(* CODESYS project SW_DMU218_3091.library
   Author: Leuze electronic GmbH + Co. KG
   Placeholder: DMU218_3091
   Title: DMU218_3091
   Version: 1.0.0
   Description: IO-Link service function blocks library
   Company: Leuze electronic GmbH + Co. KG

Project tree, tasks and I/O mapping:
  libraries: Tc2_Standard, * (Beckhoff Automation GmbH); Tc2_System, * (Beckhoff Automation GmbH); Tc2_Utilities, * (Beckhoff Automation GmbH)
  Leuze/
    DMU218_3091/
      data type ST_Leuze_IOL_AnalogRange_Data
      data type ST_Leuze_IOL_AnalogRange_Selection
      data type ST_Leuze_IOL_Commands_Data
      data type ST_Leuze_IOL_Commands_Selection
      data type ST_Leuze_IOL_Data
      data type ST_Leuze_IOL_DeviceAccessLocks_Data
      data type ST_Leuze_IOL_DeviceAccessLocks_Selection
      data type ST_Leuze_IOL_DirectParametersPage1_Data
      data type ST_Leuze_IOL_DirectParametersPage1_Selection
      data type ST_Leuze_IOL_DirectParametersPage2_Data
      data type ST_Leuze_IOL_DirectParametersPage2_Selection
      data type ST_Leuze_IOL_Network_Data
      data type ST_Leuze_IOL_Network_Selection
      data type ST_Leuze_IOL_ProcessDataLimits_Data
      data type ST_Leuze_IOL_ProcessDataLimits_Selection
      data type ST_Leuze_IOL_Selection
      data type ST_Leuze_IOL_Setpoints_Data
      data type ST_Leuze_IOL_Setpoints_Selection
      data type ST_Leuze_IOL_SwitchpointBdc1_Data
      data type ST_Leuze_IOL_SwitchpointBdc1_Selection
      data type ST_Leuze_IOL_TeachpointSp1_Data
      data type ST_Leuze_IOL_TeachpointSp1_Selection
      data type ST_Leuze_IOL_TeachpointSp2_Data
      data type ST_Leuze_IOL_TeachpointSp2_Selection
      data type ST_Leuze_IOL_TeachState_Data
      data type ST_Leuze_IOL_TeachState_Selection
    Internal/
      function F_Leuze_IOL_GetArrayT [ST]
      function F_Leuze_IOL_GetBoolean [ST]
      function F_Leuze_IOL_GetByteLength [ST]
      function F_Leuze_IOL_GetInteger [ST]
      function F_Leuze_IOL_GetRecordT [ST]
      function F_Leuze_IOL_GetString [ST]
      function F_Leuze_IOL_SetArrayT [ST]
      function F_Leuze_IOL_SetBoolean [ST]
      function F_Leuze_IOL_SetInteger [ST]
      function F_Leuze_IOL_SetRecordT [ST]
      function F_Leuze_IOL_SetString [ST]
      function F_Leuze_IOL_SortComplex [ST]
      function block FB_Leuze_IOL_AdsReadWrite [ST]
      data type ST_Leuze_IOL_CommandQueue
      data type ST_Leuze_IOL_Error
    function F_Leuze_PD_DMU218_3091 [ST]
    function block FB_Leuze_IOL_DMU218_3091 [ST]
    data type ST_Leuze_IOL_DMU218_3091
    data type ST_Leuze_PD_DMU218_3091
*)

// Leuze/DMU218_3091/ST_Leuze_IOL_AnalogRange_Data
TYPE ST_Leuze_IOL_AnalogRange_Data :
STRUCT     // [READ_WRITE]
	nLowerLimit : UINT := 150;    // [READ_WRITE]
	nUpperLimit : UINT := 1500;    // [READ_WRITE]
END_STRUCT
END_TYPE

// Leuze/DMU218_3091/ST_Leuze_IOL_AnalogRange_Selection
TYPE ST_Leuze_IOL_AnalogRange_Selection :
STRUCT     // [READ_WRITE]
	bAll : BOOL;    // [READ_WRITE] all parameters of complex data type
	bLowerLimit : BOOL;    // [READ_WRITE]
	bUpperLimit : BOOL;    // [READ_WRITE]
END_STRUCT
END_TYPE

// Leuze/DMU218_3091/ST_Leuze_IOL_Commands_Data
TYPE ST_Leuze_IOL_Commands_Data :
STRUCT     // [WRITE_ONLY] Command interface for applications. A positive acknowledge indicates the complete and correct finalization of the requested function.
	nCmdRestoreFactorySettings : UINT := 130;    // [WRITE_ONLY] Restore Factory Settings
	nCmdTeachApply : UINT := 64;    // [WRITE_ONLY] Teach Apply
	nCmdSetpoint1SingleValueTeach : UINT := 65;    // [WRITE_ONLY] Setpoint 1 Single Value Teach
	nCmdSetpoint2SingleValueTeach : UINT := 66;    // [WRITE_ONLY] Setpoint 2 Single Value Teach
	nCmdTwoValueTeachTp1Sp1 : UINT := 67;    // [WRITE_ONLY] Two Value Teach TP1 SP1
	nCmdTwoValueTeachTp2Sp1 : UINT := 68;    // [WRITE_ONLY] Two Value Teach TP2 SP1
	nCmdTwoValueTeachTp1Sp2 : UINT := 69;    // [WRITE_ONLY] Two Value Teach TP1 SP2
	nCmdTwoValueTeachTp2Sp2 : UINT := 70;    // [WRITE_ONLY] Two Value Teach TP2 SP2
	nCmdSetpoint1DynamicTeachStart : UINT := 71;    // [WRITE_ONLY] Setpoint 1 Dynamic Teach Start
	nCmdSetpoint1DynamicTeachStop : UINT := 72;    // [WRITE_ONLY] Setpoint 1 Dynamic Teach Stop
	nCmdSetpoint2DynamicTeachStart : UINT := 73;    // [WRITE_ONLY] Setpoint 2 Dynamic Teach Start
	nCmdSetpoint2DynamicTeachStop : UINT := 74;    // [WRITE_ONLY] Setpoint 2 Dynamic Teach Stop
	nCmdTeachCancel : UINT := 79;    // [WRITE_ONLY] Teach Cancel
	nCmdSetAnalogOutputLowerLimit : UINT := 161;    // [WRITE_ONLY] Set Analog Output Lower Limit
	nCmdSetAnalogOutputUpperLimit : UINT := 162;    // [WRITE_ONLY] Set Analog Output Upper Limit
	nCmdResetDiagnosisInformation : UINT := 163;    // [WRITE_ONLY] Reset Diagnosis Information
	nCmdStopMeasurement : UINT := 164;    // [WRITE_ONLY] Stop measurement
	nCmdStartMeasurement : UINT := 165;    // [WRITE_ONLY] Start measurement
	nCmdSingleMeasurement : UINT := 166;    // [WRITE_ONLY] Single measurement
	nCmdIoLink11SystemTestCommand240Event8DfeAppears : UINT := 240;    // [WRITE_ONLY] IO-Link 1.1 system test command 240, Event 8DFE appears
	nCmdIoLink11SystemTestCommand241Event8DfeDisappears : UINT := 241;    // [WRITE_ONLY] IO-Link 1.1 system test command 241, Event 8DFE disappears
	nCmdIoLink11SystemTestCommand242Event8DffAppears : UINT := 242;    // [WRITE_ONLY] IO-Link 1.1 system test command 242, Event 8DFF appears
	nCmdIoLink11SystemTestCommand243Event8DffDisappears : UINT := 243;    // [WRITE_ONLY] IO-Link 1.1 system test command 243, Event 8DFF disappears
END_STRUCT
END_TYPE

// Leuze/DMU218_3091/ST_Leuze_IOL_Commands_Selection
TYPE ST_Leuze_IOL_Commands_Selection :
STRUCT     // [WRITE_ONLY] Command interface for applications. A positive acknowledge indicates the complete and correct finalization of the requested function.
	bCmdRestoreFactorySettings : BOOL;    // [WRITE_ONLY] Restore Factory Settings
	bCmdTeachApply : BOOL;    // [WRITE_ONLY] Teach Apply
	bCmdSetpoint1SingleValueTeach : BOOL;    // [WRITE_ONLY] Setpoint 1 Single Value Teach
	bCmdSetpoint2SingleValueTeach : BOOL;    // [WRITE_ONLY] Setpoint 2 Single Value Teach
	bCmdTwoValueTeachTp1Sp1 : BOOL;    // [WRITE_ONLY] Two Value Teach TP1 SP1
	bCmdTwoValueTeachTp2Sp1 : BOOL;    // [WRITE_ONLY] Two Value Teach TP2 SP1
	bCmdTwoValueTeachTp1Sp2 : BOOL;    // [WRITE_ONLY] Two Value Teach TP1 SP2
	bCmdTwoValueTeachTp2Sp2 : BOOL;    // [WRITE_ONLY] Two Value Teach TP2 SP2
	bCmdSetpoint1DynamicTeachStart : BOOL;    // [WRITE_ONLY] Setpoint 1 Dynamic Teach Start
	bCmdSetpoint1DynamicTeachStop : BOOL;    // [WRITE_ONLY] Setpoint 1 Dynamic Teach Stop
	bCmdSetpoint2DynamicTeachStart : BOOL;    // [WRITE_ONLY] Setpoint 2 Dynamic Teach Start
	bCmdSetpoint2DynamicTeachStop : BOOL;    // [WRITE_ONLY] Setpoint 2 Dynamic Teach Stop
	bCmdTeachCancel : BOOL;    // [WRITE_ONLY] Teach Cancel
	bCmdSetAnalogOutputLowerLimit : BOOL;    // [WRITE_ONLY] Set Analog Output Lower Limit
	bCmdSetAnalogOutputUpperLimit : BOOL;    // [WRITE_ONLY] Set Analog Output Upper Limit
	bCmdResetDiagnosisInformation : BOOL;    // [WRITE_ONLY] Reset Diagnosis Information
	bCmdStopMeasurement : BOOL;    // [WRITE_ONLY] Stop measurement
	bCmdStartMeasurement : BOOL;    // [WRITE_ONLY] Start measurement
	bCmdSingleMeasurement : BOOL;    // [WRITE_ONLY] Single measurement
	bCmdIoLink11SystemTestCommand240Event8DfeAppears : BOOL;    // [WRITE_ONLY] IO-Link 1.1 system test command 240, Event 8DFE appears
	bCmdIoLink11SystemTestCommand241Event8DfeDisappears : BOOL;    // [WRITE_ONLY] IO-Link 1.1 system test command 241, Event 8DFE disappears
	bCmdIoLink11SystemTestCommand242Event8DffAppears : BOOL;    // [WRITE_ONLY] IO-Link 1.1 system test command 242, Event 8DFF appears
	bCmdIoLink11SystemTestCommand243Event8DffDisappears : BOOL;    // [WRITE_ONLY] IO-Link 1.1 system test command 243, Event 8DFF disappears
END_STRUCT
END_TYPE

// Leuze/DMU218_3091/ST_Leuze_IOL_Data
TYPE ST_Leuze_IOL_Data :
STRUCT 
	stCommands : ST_Leuze_IOL_Commands_Data;
	stDirectParametersPage1 : ST_Leuze_IOL_DirectParametersPage1_Data;
	stDirectParametersPage2 : ST_Leuze_IOL_DirectParametersPage2_Data;
	nSystemCommand : UINT;    // [WRITE_ONLY] Command interface for applications. A positive acknowledge indicates the complete and correct finalization of the requested function.
	stDeviceAccessLocks : ST_Leuze_IOL_DeviceAccessLocks_Data;
	sVendorName : STRING := 'Leuze electronic GmbH + Co. KG';    // [READ_ONLY] The vendor name that is assigned to a Vendor ID.
	sVendorText : STRING := 'The Sensor People';    // [READ_ONLY] Additional information about the vendor.
	sProductName : STRING;    // [READ_ONLY] Complete product name.
	sProductId : STRING;    // [READ_ONLY] Vendor-specific product or type identification (e.g., item number or model number).
	sProductText : STRING;    // [READ_ONLY] Additional product information for the device.
	sFirmwareRevision : STRING;    // [READ_ONLY] Unique, vendor-specific identifier of the firmware revision of the individual device.
	sApplicationSpecificTag : STRING;    // [READ_WRITE] Possibility to mark a device with user- or application-specific information.
	nErrorCount : UINT;    // [READ_ONLY] Number of errors that occurred in the technology-specific application since power on or restart.
	nDeviceStatus : UINT;    // [READ_ONLY] Indicator for the current device condition and diagnosis state.
	stTeachState : ST_Leuze_IOL_TeachState_Data;
	stSetpoints : ST_Leuze_IOL_Setpoints_Data;
	stSwitchpointBdc1 : ST_Leuze_IOL_SwitchpointBdc1_Data;
	sLot : STRING;    // [READ_ONLY] production lot
	nOnDelaySwitchingOutput : UINT := 0;    // [READ_WRITE] on delay for the binary data channel
	nOffDelaySwitchingOutput : UINT := 0;    // [READ_WRITE] off delay for the binary data channel
	nMultiIOPin4 : UINT := 0;    // [READ_WRITE] polarity of the switching output
	nMultiIOPin2 : UINT := 2;    // [READ_WRITE] operation mode for Multi I/O (Pin 2)
	stAnalogRange : ST_Leuze_IOL_AnalogRange_Data;
	nTemperatureCompensation : UINT := 0;    // [READ_WRITE]
	stTeachpointSp1 : ST_Leuze_IOL_TeachpointSp1_Data;
	stTeachpointSp2 : ST_Leuze_IOL_TeachpointSp2_Data;
	stProcessDataLimits : ST_Leuze_IOL_ProcessDataLimits_Data;
	nSwitchCounter : UINT := 0;    // [READ_ONLY] number of switching after power-up or reset
	nTemperatureInternal : INT;    // [READ_ONLY] Sensor temperature
	stNetwork : ST_Leuze_IOL_Network_Data;
END_STRUCT
END_TYPE

// Leuze/DMU218_3091/ST_Leuze_IOL_DeviceAccessLocks_Data
TYPE ST_Leuze_IOL_DeviceAccessLocks_Data :
STRUCT     // [READ_WRITE] The access to the device parameters can be restricted by setting appropriate flags within this parameter.
	bParameterWriteAccess : BOOL := 0;    // [READ_WRITE] This lock prevents the write access to all read/write parameters of the device except for the parameter 'Device Access Locks'.
	bDataStorage : BOOL;    // [READ_WRITE] This lock prevents the write access to the device parameters via the data storage mechanism.
	bLocalParameterization : BOOL := 0;    // [READ_WRITE] This lock prevents the device settings from being changed via local operating elements on the device.
	bLocalUserInterface : BOOL;    // [READ_WRITE] This lock prevents the access to the device settings and display via a local user interface. The user interface is disabled.
END_STRUCT
END_TYPE

// Leuze/DMU218_3091/ST_Leuze_IOL_DeviceAccessLocks_Selection
TYPE ST_Leuze_IOL_DeviceAccessLocks_Selection :
STRUCT     // [READ_WRITE] The access to the device parameters can be restricted by setting appropriate flags within this parameter.
	bAll : BOOL;    // [READ_WRITE] all parameters of complex data type
END_STRUCT
END_TYPE

// Leuze/DMU218_3091/ST_Leuze_IOL_DirectParametersPage1_Data
TYPE ST_Leuze_IOL_DirectParametersPage1_Data :
STRUCT     // [READ_WRITE] Comprises the required parameters defining the communication characteristics and identifiers for device validation.
	nReserved_1 : UINT;    // [READ_ONLY] ; Suffix "_1" (parameter index or subindex) added because of duplicate parameter names.
	nMasterCycleTime : UINT;    // [READ_ONLY] Communication: Current communication cycle duration used by the master. This value defines the process data cycle.
	nMinCycleTime : UINT;    // [READ_ONLY] Communication: Minimum communication cycle duration supported by the device. This value defines the lowest possible process data cycle.
	nMSequenceCapability : UINT;    // [READ_ONLY] Communication: Information on the structure and the supported features of the communication messages.
	nIoLinkRevisionId : UINT := 17;    // [READ_ONLY] Communication: Identifier for the currently used communication protocol revision.
	nProcessDataInputLength : UINT;    // [READ_ONLY] Communication: Information on width and features of the process input data (Process Data from Device to Master).
	nProcessDataOutputLength : UINT;    // [READ_ONLY] Communication: Information on width of the process output data (Process Data from Master to Device).
	nVendorId1 : UINT;    // [READ_ONLY] Identification: Highest octet of the Vendor ID. Combined with the parameter Vendor ID 2, this parameter defines the 16-bit value of the unique Vendor ID as assigned by the IO-Link Community.
	nVendorId2 : UINT;    // [READ_ONLY] Identification: Lowest octet of the Vendor ID. Combined with the parameter Vendor ID 1, this parameter defines the 16-bit value of the unique Vendor ID as assigned by the IO-Link Community.
	nDeviceId1 : UINT;    // [READ_ONLY] Identification: Highest octet of the Device ID. Combined with the parameters Device ID 2 and 3, this parameter defines the 24-bit value of the vendor-specific Device ID.
	nDeviceId2 : UINT;    // [READ_ONLY] Identification: Middle octet of the Device ID. Combined with the parameters Device ID 1 and 3, this parameter defines the 24-bit value of the vendor-specific Device ID.
	nDeviceId3 : UINT;    // [READ_ONLY] Identification: Lowest octet of the Device ID. Combined with the parameters Device ID 1 and 2, this parameter defines the 24-bit value of the vendor-specific Device ID.
	nReserved_13 : UINT;    // [READ_ONLY] ; Suffix "_13" (parameter index or subindex) added because of duplicate parameter names.
	nReserved_14 : UINT;    // [READ_ONLY] ; Suffix "_14" (parameter index or subindex) added because of duplicate parameter names.
	nReserved_15 : UINT;    // [READ_ONLY] ; Suffix "_15" (parameter index or subindex) added because of duplicate parameter names.
	nSystemCommand : UINT;    // [WRITE_ONLY] Application: Command interface for devices without ISDU support. Validity and execution of commands are not confirmed.
END_STRUCT
END_TYPE

// Leuze/DMU218_3091/ST_Leuze_IOL_DirectParametersPage1_Selection
TYPE ST_Leuze_IOL_DirectParametersPage1_Selection :
STRUCT     // [READ_WRITE] Comprises the required parameters defining the communication characteristics and identifiers for device validation.
	bAll : BOOL;    // [READ_WRITE] all parameters of complex data type
	bReserved_1 : BOOL;    // [READ_ONLY] ; Suffix "_1" (parameter index or subindex) added because of duplicate parameter names.
	bMasterCycleTime : BOOL;    // [READ_ONLY] Communication: Current communication cycle duration used by the master. This value defines the process data cycle.
	bMinCycleTime : BOOL;    // [READ_ONLY] Communication: Minimum communication cycle duration supported by the device. This value defines the lowest possible process data cycle.
	bMSequenceCapability : BOOL;    // [READ_ONLY] Communication: Information on the structure and the supported features of the communication messages.
	bIoLinkRevisionId : BOOL;    // [READ_ONLY] Communication: Identifier for the currently used communication protocol revision.
	bProcessDataInputLength : BOOL;    // [READ_ONLY] Communication: Information on width and features of the process input data (Process Data from Device to Master).
	bProcessDataOutputLength : BOOL;    // [READ_ONLY] Communication: Information on width of the process output data (Process Data from Master to Device).
	bVendorId1 : BOOL;    // [READ_ONLY] Identification: Highest octet of the Vendor ID. Combined with the parameter Vendor ID 2, this parameter defines the 16-bit value of the unique Vendor ID as assigned by the IO-Link Community.
	bVendorId2 : BOOL;    // [READ_ONLY] Identification: Lowest octet of the Vendor ID. Combined with the parameter Vendor ID 1, this parameter defines the 16-bit value of the unique Vendor ID as assigned by the IO-Link Community.
	bDeviceId1 : BOOL;    // [READ_ONLY] Identification: Highest octet of the Device ID. Combined with the parameters Device ID 2 and 3, this parameter defines the 24-bit value of the vendor-specific Device ID.
	bDeviceId2 : BOOL;    // [READ_ONLY] Identification: Middle octet of the Device ID. Combined with the parameters Device ID 1 and 3, this parameter defines the 24-bit value of the vendor-specific Device ID.
	bDeviceId3 : BOOL;    // [READ_ONLY] Identification: Lowest octet of the Device ID. Combined with the parameters Device ID 1 and 2, this parameter defines the 24-bit value of the vendor-specific Device ID.
	bReserved_13 : BOOL;    // [READ_ONLY] ; Suffix "_13" (parameter index or subindex) added because of duplicate parameter names.
	bReserved_14 : BOOL;    // [READ_ONLY] ; Suffix "_14" (parameter index or subindex) added because of duplicate parameter names.
	bReserved_15 : BOOL;    // [READ_ONLY] ; Suffix "_15" (parameter index or subindex) added because of duplicate parameter names.
	bSystemCommand : BOOL;    // [WRITE_ONLY] Application: Command interface for devices without ISDU support. Validity and execution of commands are not confirmed.
END_STRUCT
END_TYPE

// Leuze/DMU218_3091/ST_Leuze_IOL_DirectParametersPage2_Data
TYPE ST_Leuze_IOL_DirectParametersPage2_Data :
STRUCT     // [READ_WRITE] A set of parameters for devices without ISDU support.
	nDeviceSpecificParameter1 : UINT;    // [READ_WRITE]
	nDeviceSpecificParameter2 : UINT;    // [READ_WRITE]
	nDeviceSpecificParameter3 : UINT;    // [READ_WRITE]
	nDeviceSpecificParameter4 : UINT;    // [READ_WRITE]
	nDeviceSpecificParameter5 : UINT;    // [READ_WRITE]
	nDeviceSpecificParameter6 : UINT;    // [READ_WRITE]
	nDeviceSpecificParameter7 : UINT;    // [READ_WRITE]
	nDeviceSpecificParameter8 : UINT;    // [READ_WRITE]
	nDeviceSpecificParameter9 : UINT;    // [READ_WRITE]
	nDeviceSpecificParameter10 : UINT;    // [READ_WRITE]
	nDeviceSpecificParameter11 : UINT;    // [READ_WRITE]
	nDeviceSpecificParameter12 : UINT;    // [READ_WRITE]
	nDeviceSpecificParameter13 : UINT;    // [READ_WRITE]
	nDeviceSpecificParameter14 : UINT;    // [READ_WRITE]
	nDeviceSpecificParameter15 : UINT;    // [READ_WRITE]
	nDeviceSpecificParameter16 : UINT;    // [READ_WRITE]
END_STRUCT
END_TYPE

// Leuze/DMU218_3091/ST_Leuze_IOL_DirectParametersPage2_Selection
TYPE ST_Leuze_IOL_DirectParametersPage2_Selection :
STRUCT     // [READ_WRITE] A set of parameters for devices without ISDU support.
	bAll : BOOL;    // [READ_WRITE] all parameters of complex data type
	bDeviceSpecificParameter1 : BOOL;    // [READ_WRITE]
	bDeviceSpecificParameter2 : BOOL;    // [READ_WRITE]
	bDeviceSpecificParameter3 : BOOL;    // [READ_WRITE]
	bDeviceSpecificParameter4 : BOOL;    // [READ_WRITE]
	bDeviceSpecificParameter5 : BOOL;    // [READ_WRITE]
	bDeviceSpecificParameter6 : BOOL;    // [READ_WRITE]
	bDeviceSpecificParameter7 : BOOL;    // [READ_WRITE]
	bDeviceSpecificParameter8 : BOOL;    // [READ_WRITE]
	bDeviceSpecificParameter9 : BOOL;    // [READ_WRITE]
	bDeviceSpecificParameter10 : BOOL;    // [READ_WRITE]
	bDeviceSpecificParameter11 : BOOL;    // [READ_WRITE]
	bDeviceSpecificParameter12 : BOOL;    // [READ_WRITE]
	bDeviceSpecificParameter13 : BOOL;    // [READ_WRITE]
	bDeviceSpecificParameter14 : BOOL;    // [READ_WRITE]
	bDeviceSpecificParameter15 : BOOL;    // [READ_WRITE]
	bDeviceSpecificParameter16 : BOOL;    // [READ_WRITE]
END_STRUCT
END_TYPE

// Leuze/DMU218_3091/ST_Leuze_IOL_Network_Data
TYPE ST_Leuze_IOL_Network_Data :
STRUCT     // [READ_WRITE]
	nRoleInNetwork : UINT := 0;    // [READ_WRITE]
	nDeviceNoMasterHighestNo : UINT := 1;    // [READ_WRITE]
END_STRUCT
END_TYPE

// Leuze/DMU218_3091/ST_Leuze_IOL_Network_Selection
TYPE ST_Leuze_IOL_Network_Selection :
STRUCT     // [READ_WRITE]
	bAll : BOOL;    // [READ_WRITE] all parameters of complex data type
	bRoleInNetwork : BOOL;    // [READ_WRITE]
	bDeviceNoMasterHighestNo : BOOL;    // [READ_WRITE]
END_STRUCT
END_TYPE

// Leuze/DMU218_3091/ST_Leuze_IOL_ProcessDataLimits_Data
TYPE ST_Leuze_IOL_ProcessDataLimits_Data :
STRUCT     // [READ_ONLY] Process data limit values
	nLower : UINT;    // [READ_ONLY] lower limit after power-up or reset
	nUpper : UINT;    // [READ_ONLY] upper limit after power-up or reset
END_STRUCT
END_TYPE

// Leuze/DMU218_3091/ST_Leuze_IOL_ProcessDataLimits_Selection
TYPE ST_Leuze_IOL_ProcessDataLimits_Selection :
STRUCT     // [READ_ONLY] Process data limit values
	bAll : BOOL;    // [READ_ONLY] all parameters of complex data type
	bLower : BOOL;    // [READ_ONLY] lower limit after power-up or reset
	bUpper : BOOL;    // [READ_ONLY] upper limit after power-up or reset
END_STRUCT
END_TYPE

// Leuze/DMU218_3091/ST_Leuze_IOL_Selection
TYPE ST_Leuze_IOL_Selection :
STRUCT 
	stCommands : ST_Leuze_IOL_Commands_Selection;
	stDirectParametersPage1 : ST_Leuze_IOL_DirectParametersPage1_Selection;
	stDirectParametersPage2 : ST_Leuze_IOL_DirectParametersPage2_Selection;
	bSystemCommand : BOOL;    // [WRITE_ONLY] Command interface for applications. A positive acknowledge indicates the complete and correct finalization of the requested function.
	stDeviceAccessLocks : ST_Leuze_IOL_DeviceAccessLocks_Selection;
	bVendorName : BOOL;    // [READ_ONLY] The vendor name that is assigned to a Vendor ID.
	bVendorText : BOOL;    // [READ_ONLY] Additional information about the vendor.
	bProductName : BOOL;    // [READ_ONLY] Complete product name.
	bProductId : BOOL;    // [READ_ONLY] Vendor-specific product or type identification (e.g., item number or model number).
	bProductText : BOOL;    // [READ_ONLY] Additional product information for the device.
	bFirmwareRevision : BOOL;    // [READ_ONLY] Unique, vendor-specific identifier of the firmware revision of the individual device.
	bApplicationSpecificTag : BOOL;    // [READ_WRITE] Possibility to mark a device with user- or application-specific information.
	bErrorCount : BOOL;    // [READ_ONLY] Number of errors that occurred in the technology-specific application since power on or restart.
	bDeviceStatus : BOOL;    // [READ_ONLY] Indicator for the current device condition and diagnosis state.
	stTeachState : ST_Leuze_IOL_TeachState_Selection;
	stSetpoints : ST_Leuze_IOL_Setpoints_Selection;
	stSwitchpointBdc1 : ST_Leuze_IOL_SwitchpointBdc1_Selection;
	bLot : BOOL;    // [READ_ONLY] production lot
	bOnDelaySwitchingOutput : BOOL;    // [READ_WRITE] on delay for the binary data channel
	bOffDelaySwitchingOutput : BOOL;    // [READ_WRITE] off delay for the binary data channel
	bMultiIOPin4 : BOOL;    // [READ_WRITE] polarity of the switching output
	bMultiIOPin2 : BOOL;    // [READ_WRITE] operation mode for Multi I/O (Pin 2)
	stAnalogRange : ST_Leuze_IOL_AnalogRange_Selection;
	bTemperatureCompensation : BOOL;    // [READ_WRITE]
	stTeachpointSp1 : ST_Leuze_IOL_TeachpointSp1_Selection;
	stTeachpointSp2 : ST_Leuze_IOL_TeachpointSp2_Selection;
	stProcessDataLimits : ST_Leuze_IOL_ProcessDataLimits_Selection;
	bSwitchCounter : BOOL;    // [READ_ONLY] number of switching after power-up or reset
	bTemperatureInternal : BOOL;    // [READ_ONLY] Sensor temperature
	stNetwork : ST_Leuze_IOL_Network_Selection;
END_STRUCT
END_TYPE

// Leuze/DMU218_3091/ST_Leuze_IOL_Setpoints_Data
TYPE ST_Leuze_IOL_Setpoints_Data :
STRUCT     // [READ_WRITE] threshold measurement value of a sensor for the edge of a binary output signal 1
	nParam1Bdc1Q1 : UINT := 150;    // [READ_WRITE] threshold measurement value
	nParam2Bdc1Q1 : UINT := 1500;    // [READ_WRITE] threshold measurement value
END_STRUCT
END_TYPE

// Leuze/DMU218_3091/ST_Leuze_IOL_Setpoints_Selection
TYPE ST_Leuze_IOL_Setpoints_Selection :
STRUCT     // [READ_WRITE] threshold measurement value of a sensor for the edge of a binary output signal 1
	bAll : BOOL;    // [READ_WRITE] all parameters of complex data type
	bParam1Bdc1Q1 : BOOL;    // [READ_WRITE] threshold measurement value
	bParam2Bdc1Q1 : BOOL;    // [READ_WRITE] threshold measurement value
END_STRUCT
END_TYPE

// Leuze/DMU218_3091/ST_Leuze_IOL_SwitchpointBdc1_Data
TYPE ST_Leuze_IOL_SwitchpointBdc1_Data :
STRUCT     // [READ_WRITE] mode, logic and hysteresis for binary data channel 1
	nLogic : UINT := 0;    // [READ_WRITE] switching information is transmitted in inverted or not inverted manner
	nMode : UINT := 2;    // [READ_WRITE] operation mode for binary signal
	nHysteresis : UINT := 2;    // [READ_WRITE]
END_STRUCT
END_TYPE

// Leuze/DMU218_3091/ST_Leuze_IOL_SwitchpointBdc1_Selection
TYPE ST_Leuze_IOL_SwitchpointBdc1_Selection :
STRUCT     // [READ_WRITE] mode, logic and hysteresis for binary data channel 1
	bAll : BOOL;    // [READ_WRITE] all parameters of complex data type
	bLogic : BOOL;    // [READ_WRITE] switching information is transmitted in inverted or not inverted manner
	bMode : BOOL;    // [READ_WRITE] operation mode for binary signal
	bHysteresis : BOOL;    // [READ_WRITE]
END_STRUCT
END_TYPE

// Leuze/DMU218_3091/ST_Leuze_IOL_TeachpointSp1_Data
TYPE ST_Leuze_IOL_TeachpointSp1_Data :
STRUCT     // [READ_ONLY] Values detected during teach
	nTp1 : UINT;    // [READ_ONLY] detected lower limit during teach-in procedure
	nTp2 : UINT;    // [READ_ONLY] detected upper limit during teach-in procedure
END_STRUCT
END_TYPE

// Leuze/DMU218_3091/ST_Leuze_IOL_TeachpointSp1_Selection
TYPE ST_Leuze_IOL_TeachpointSp1_Selection :
STRUCT     // [READ_ONLY] Values detected during teach
	bAll : BOOL;    // [READ_ONLY] all parameters of complex data type
	bTp1 : BOOL;    // [READ_ONLY] detected lower limit during teach-in procedure
	bTp2 : BOOL;    // [READ_ONLY] detected upper limit during teach-in procedure
END_STRUCT
END_TYPE

// Leuze/DMU218_3091/ST_Leuze_IOL_TeachpointSp2_Data
TYPE ST_Leuze_IOL_TeachpointSp2_Data :
STRUCT     // [READ_ONLY] Values detected during teach
	nTp1 : UINT;    // [READ_ONLY] detected lower limit during teach-in procedure
	nTp2 : UINT;    // [READ_ONLY] detected upper limit during teach-in procedure
END_STRUCT
END_TYPE

// Leuze/DMU218_3091/ST_Leuze_IOL_TeachpointSp2_Selection
TYPE ST_Leuze_IOL_TeachpointSp2_Selection :
STRUCT     // [READ_ONLY] Values detected during teach
	bAll : BOOL;    // [READ_ONLY] all parameters of complex data type
	bTp1 : BOOL;    // [READ_ONLY] detected lower limit during teach-in procedure
	bTp2 : BOOL;    // [READ_ONLY] detected upper limit during teach-in procedure
END_STRUCT
END_TYPE

// Leuze/DMU218_3091/ST_Leuze_IOL_TeachState_Data
TYPE ST_Leuze_IOL_TeachState_Data :
STRUCT     // [READ_ONLY] indication of the current state of the teach-in procedure and teach point setting
	nTeachState : UINT := 0;    // [READ_ONLY] indication of the current state of the teach-in procedure
END_STRUCT
END_TYPE

// Leuze/DMU218_3091/ST_Leuze_IOL_TeachState_Selection
TYPE ST_Leuze_IOL_TeachState_Selection :
STRUCT     // [READ_ONLY] indication of the current state of the teach-in procedure and teach point setting
	bAll : BOOL;    // [READ_ONLY] all parameters of complex data type
END_STRUCT
END_TYPE

// Leuze/Internal/ST_Leuze_IOL_CommandQueue
TYPE ST_Leuze_IOL_CommandQueue :
STRUCT
	nIndex : INT;		// Index of parameter in queue
    nSubIndex : INT;	// SubIndex of a parameter in queue
    nBitLength : UINT;	// Bit length of a parameter
END_STRUCT
END_TYPE

// Leuze/Internal/ST_Leuze_IOL_Error
TYPE ST_Leuze_IOL_Error :
STRUCT
    nBlockError : WORD;			// Error number representing FB where error occured 
	nAdsReadError : UDINT;		// ADS read error code
	nAdsWriteError : UDINT;		// ADS write error code
	nIndex : INT;				// IO-Link index to which the error code refers
	nSubIndex : INT;			// IO-Link sub-index to which the error code refers
END_STRUCT
END_TYPE

// Leuze/ST_Leuze_IOL_DMU218_3091
TYPE ST_Leuze_IOL_DMU218_3091 :
STRUCT
	stSelection : ST_Leuze_IOL_Selection;
	stData : ST_Leuze_IOL_Data;
END_STRUCT
END_TYPE

// Leuze/ST_Leuze_PD_DMU218_3091
TYPE ST_Leuze_PD_DMU218_3091 :
STRUCT
	nMeasuredValue : UINT;
	bSwitchStateBdc1Q1 : BOOL;
END_STRUCT
END_TYPE

// Leuze/Internal/F_Leuze_IOL_GetArrayT
FUNCTION F_Leuze_IOL_GetArrayT : BOOL
VAR_INPUT
	nArraySize : UINT;
    nItemPosition : UINT;
    nBitLength : UINT;
END_VAR
VAR_IN_OUT 
      aIolRecords : ARRAY[0..cNUMBER_IOLINK_DATA] OF BYTE;
      aTempItems : ARRAY[0..cNUMBER_IOLINK_DATA] OF BYTE;
END_VAR
VAR
      nTempArrayByteLength : UINT;
      nTempStartByte : UINT;
      nTempStartBit : UINT;
      nTempIolBitLength : UINT;
      nTempIolByteLength : UINT;
      nTempIndex : UINT;
      nTempShiftByte : BYTE;
      bTempByteFill : BOOL;
END_VAR
VAR CONSTANT 
	  cNUMBER_IOLINK_DATA : UINT := 255;   //   Number of IO Link record data
	  cBITS_IN_BYTE : UINT := 8;   //   Number of bits in byte
END_VAR

// =============================================================================
// Name:    IO-Link internal function 
//          Array data type - Integer, Bool
// Date:    01.01.2021
// ==============================================================================

// Initialize variables
	bTempByteFill := FALSE;
	
// Bit length of the current item
	nTempIolBitLength := nBitLength;
	
// Get byte length of the current item
	nTempIolByteLength := F_Leuze_IOL_GetByteLength(nTempIolBitLength);
	
// Get byte length of the whole array
	nTempArrayByteLength := F_Leuze_IOL_GetByteLength(nArraySize);
	
	
// Calculate the start byte of the current array item
	nTempStartByte := nTempArrayByteLength - 1 - ((nArraySize - (nItemPosition * nTempIolBitLength)) / cBITS_IN_BYTE);
	
// Calculate the start bit of the current array item
	nTempStartBit := (nArraySize - (nItemPosition * nTempIolBitLength)) MOD cBITS_IN_BYTE;
	
// Calculate index
	nTempIndex := nTempIolByteLength - 1;
	
// Get array item
	WHILE nTempIolBitLength > 0 DO
		IF NOT bTempByteFill THEN	    
			IF (nTempIolBitLength + nTempStartBit) < cBITS_IN_BYTE THEN
				nTempShiftByte := SHL(aIolRecords[nTempStartByte], cBITS_IN_BYTE - (nTempIolBitLength + nTempStartBit));
				nTempShiftByte := SHR(nTempShiftByte, cBITS_IN_BYTE - nTempIolBitLength);
			ELSE
				nTempShiftByte := SHR(aIolRecords[nTempStartByte], nTempStartBit);
			END_IF;
			
			aTempItems[nTempIndex] := nTempShiftByte;
			
			IF (nTempStartBit + nTempIolBitLength) = cBITS_IN_BYTE THEN
				nTempStartByte := nTempStartByte - 1;
			END_IF;
			
			IF (nTempStartBit + nTempIolBitLength) > cBITS_IN_BYTE THEN
				nTempStartByte := nTempStartByte - 1;
				bTempByteFill := TRUE;
			ELSE
				nTempIndex := nTempIndex - 1;
			END_IF;
			
			nTempIolBitLength := nTempIolBitLength - (cBITS_IN_BYTE - nTempStartBit);
		ELSE	   
	    IF nTempStartBit >= nTempIolBitLength THEN
			nTempShiftByte := SHL(aIolRecords[nTempStartByte], cBITS_IN_BYTE - nTempIolBitLength);
			nTempShiftByte := SHR(nTempShiftByte, nTempStartBit - nTempIolBitLength);
	    ELSE
	    	nTempShiftByte := SHL(aIolRecords[nTempStartByte], cBITS_IN_BYTE - nTempStartBit);
	    END_IF;
	    
	    aTempItems[nTempIndex] := nTempShiftByte XOR aTempItems[nTempIndex];	    
	    nTempIolBitLength := nTempIolBitLength - nTempStartBit;
	    nTempIndex := nTempIndex - 1;
	    bTempByteFill := FALSE;
		END_IF;
	END_WHILE;

END_FUNCTION

// Leuze/Internal/F_Leuze_IOL_GetByteLength
FUNCTION F_Leuze_IOL_GetByteLength : UINT
VAR_INPUT
	nBitLength: UINT;
END_VAR
VAR
	nByteLength: UINT;
END_VAR

VAR CONSTANT
	cBITS_IN_BYTE: UINT := 8;
END_VAR

nByteLength := nBitLength / cBITS_IN_BYTE;
IF NOT (nBitLength MOD cBITS_IN_BYTE = 0) THEN
		nByteLength := nByteLength + 1;
END_IF;
F_Leuze_IOL_GetByteLength := nByteLength;

END_FUNCTION

// Leuze/Internal/F_Leuze_IOL_GetBoolean
FUNCTION F_Leuze_IOL_GetBoolean : BOOL
VAR_INPUT 
      nComplex : INT;	// Data type: cBASIC_TYPE, cCOMPLEX_RECORD_TYPE, cCOMPLEX_ARRAY_TYPE
      nComplexDataTypeSize : INT;	// Record or Array type size
      nOffset : INT;	// Bit Offset
   END_VAR
   VAR_IN_OUT 
      aIolRecords : ARRAY[0..cNUMBER_IOLINK_DATA] OF BYTE;
      aTempItems : ARRAY[0..cNUMBER_IOLINK_DATA] OF BYTE;
   END_VAR
   VAR CONSTANT 
      cNUMBER_IOLINK_DATA : INT := 255;   //   Number of IO Link record data
      cBASIC_TYPE : INT := 0;
      cCOMPLEX_RECORD_TYPE : INT := 1;
      cCOMPLEX_ARRAY_TYPE : INT := 2;
   END_VAR

// =============================================================================
// Name:    IO-Link internal function 
//  		GetBoolean
// Date:    01.07.2020
// ==============================================================================
	
// Data type is part of a Record data type
IF nComplex = cCOMPLEX_RECORD_TYPE THEN		
  F_Leuze_IOL_GetRecordT(nComplexDataTypeSize, nOffset, 1, aIolRecords, aTempItems);
  // Data type is part of a Array data type
ELSIF nComplex = cCOMPLEX_ARRAY_TYPE THEN
  F_Leuze_IOL_GetArrayT(INT_TO_UINT(nComplexDataTypeSize), INT_TO_UINT(nOffset), 1, aIolRecords, aTempItems);
END_IF;
	
// In a nComplex data type the coding of booleans are only 1 bit wide. There is no padding to byte 
IF nComplex > cBASIC_TYPE THEN
  IF aTempItems[0].0 = 1 THEN
    F_Leuze_IOL_GetBoolean := TRUE;
  ELSE
    F_Leuze_IOL_GetBoolean := FALSE;
  END_IF;
ELSE
  IF aIolRecords[0] > 16#00 THEN
    F_Leuze_IOL_GetBoolean := TRUE;
  ELSE
    F_Leuze_IOL_GetBoolean := FALSE;
  END_IF;
END_IF;

END_FUNCTION

// Leuze/Internal/F_Leuze_IOL_GetRecordT
FUNCTION F_Leuze_IOL_GetRecordT : BOOL
VAR_INPUT 
      nRecordSize : INT;
      nBitOffset : INT;
      nBitLength : INT;
   END_VAR
   VAR_IN_OUT 
      aIolRecords : ARRAY[0..cNUMBER_IOLINK_DATA] OF BYTE;
      aTempItems : ARRAY[0..cNUMBER_IOLINK_DATA] OF BYTE;
   END_VAR
   VAR
      nTempStartByte : INT;
      nTempStartBit : Int;
      tempIOLBitLength : Int;
      tempIOLByteLength : Int;
      nTempIndex : Int;
      nTempShiftByte : Byte;
      bTempByteFill : Bool;
   END_VAR
   VAR CONSTANT 
	  cNUMBER_IOLINK_DATA : INT := 255;   //   Number of IO Link record data
	  cBITS_IN_BYTE : INT := 8;   //   Number of bits in byte
   END_VAR

// =============================================================================
// Name:    IO-Link internal function 
//    		Record data type - Integer, Bool
// Date:    01.07.2020
// ==============================================================================
	
// Initialize variables
	bTempByteFill := FALSE;
	
// Bit length of the current item
	tempIOLBitLength := nBitLength;
	
// Get byte length of the current item
	tempIOLByteLength := tempIOLBitLength / cBITS_IN_BYTE;
	IF NOT (tempIOLBitLength MOD cBITS_IN_BYTE = 0) THEN
		tempIOLByteLength := tempIOLByteLength + 1;
	END_IF;
		
// Calculate the start byte of the current item
	nTempStartByte := (nRecordSize / cBITS_IN_BYTE) - 1 - (nBitOffset / cBITS_IN_BYTE);
	IF NOT(nRecordSize MOD cBITS_IN_BYTE = 0) THEN
		nTempStartByte := nTempStartByte +1;
	END_IF;

// Calculate the start bit of the current item
	nTempStartBit := nBitOffset MOD cBITS_IN_BYTE;
	
// Calculate index
	nTempIndex := tempIOLByteLength - 1;
	
// Get record item
	WHILE tempIOLBitLength > 0 DO
		IF NOT bTempByteFill THEN		
			IF (tempIOLBitLength + nTempStartBit) < cBITS_IN_BYTE THEN
				nTempShiftByte := SHL(aIolRecords[nTempStartByte], INT_TO_UINT(cBITS_IN_BYTE - (tempIOLBitLength + nTempStartBit)));
				nTempShiftByte := SHR(nTempShiftByte, INT_TO_UINT(cBITS_IN_BYTE - tempIOLBitLength));
			ELSE
				nTempShiftByte := SHR(aIolRecords[nTempStartByte], INT_TO_UINT(nTempStartBit));
			END_IF;
			aTempItems[nTempIndex] := nTempShiftByte;
			
			IF (nTempStartBit + tempIOLBitLength) = cBITS_IN_BYTE THEN
				nTempStartByte := nTempStartByte - 1;
			END_IF;
			
			IF (nTempStartBit + tempIOLBitLength) > cBITS_IN_BYTE THEN
				nTempStartByte := nTempStartByte - 1;
				bTempByteFill := TRUE;
			ELSE
				nTempIndex := nTempIndex - 1;
			END_IF;
			
			tempIOLBitLength := tempIOLBitLength - (cBITS_IN_BYTE - nTempStartBit);
		ELSE		
			IF nTempStartBit >= tempIOLBitLength THEN
				nTempShiftByte := SHL(aIolRecords[nTempStartByte], INT_TO_UINT(cBITS_IN_BYTE - tempIOLBitLength));
				nTempShiftByte := SHR(nTempShiftByte, INT_TO_UINT(nTempStartBit - tempIOLBitLength));
			ELSE
				nTempShiftByte := SHL(aIolRecords[nTempStartByte], INT_TO_UINT(cBITS_IN_BYTE - nTempStartBit));
			END_IF;			
			aTempItems[nTempIndex] := nTempShiftByte XOR aTempItems[nTempIndex];			
			tempIOLBitLength := tempIOLBitLength - nTempStartBit;
			nTempIndex := nTempIndex - 1;
			bTempByteFill := FALSE;
		END_IF;
	END_WHILE;

END_FUNCTION

// Leuze/Internal/F_Leuze_IOL_GetInteger
FUNCTION F_Leuze_IOL_GetInteger : DWORD
VAR_INPUT 
      nComplex : INT;	// Data type: cBASIC_TYPE, cCOMPLEX_RECORD_TYPE, cCOMPLEX_ARRAY_TYPE
      nComplexDataTypeSize : INT;	// Record or Array type size
      nOffset : INT;	// Bit Offset
      nBitLength : INT;
      bIsSigned : BOOL;
   END_VAR
   VAR_IN_OUT 
      aIolRecords : ARRAY[0..cNUMBER_IOLINK_DATA] OF BYTE;
      aTempItems : ARRAY[0..cNUMBER_IOLINK_DATA] OF BYTE;
   END_VAR
VAR
	nTempOutput : DWORD;   
    nTempIndex : INT;
    nTempIolByteLength : INT;
    nTemp : DWORD;
    aTempValues : ARRAY[0..3] OF BYTE;
	pOutput: POINTER TO ARRAY[0..3] OF BYTE;
END_VAR
VAR CONSTANT
	  cNUMBER_IOLINK_DATA : INT := 255;   //   Number of IO Link record data
	  cBITS_IN_BYTE : INT := 8;   //   Number of bits in byte
      cBASIC_TYPE : INT := 0;
      cCOMPLEX_RECORD_TYPE : INT := 1;
      cCOMPLEX_ARRAY_TYPE : INT := 2;
   END_VAR

// =============================================================================
// Name:    IO-Link internal function 
//   		GetInteger
// Date:    01.01.2021
// ==============================================================================

// Data type is part of a Record data type
	IF nComplex = cCOMPLEX_RECORD_TYPE THEN
		F_Leuze_IOL_GetRecordT(nComplexDataTypeSize, nOffset, nBitLength, aIolRecords, aTempItems);
	// Data type is part of a Array data type
	ELSIF nComplex = cCOMPLEX_ARRAY_TYPE THEN
		F_Leuze_IOL_GetArrayT(INT_TO_UINT(nComplexDataTypeSize), INT_TO_UINT(nOffset), INT_TO_UINT(nBitLength), aIolRecords, aTempItems);
	END_IF;
	
// Initialization
	F_Leuze_IOL_GetInteger := 16#00;
	aTempValues[0] := 0;
	aTempValues[1] := 0;
	aTempValues[2] := 0;
	aTempValues[3] := 0;
	
// Get byte length
	nTempIolByteLength := nBitLength / cBITS_IN_BYTE;
	IF NOT (nBitLength MOD cBITS_IN_BYTE = 0) THEN
		nTempIolByteLength := nTempIolByteLength + 1;
	END_IF;
	
// There is no padding to 1,2,4 byte if a nComplex data type is used
	IF (nComplex = cBASIC_TYPE) AND (nTempIolByteLength = 3) THEN
		nTempIolByteLength := 4;
	END_IF;
	
	IF nTempIolByteLength > 0 AND nTempIolByteLength <= 4 THEN
	// Get the value out of the IO-Link Record and change the byte order
	FOR nTempIndex := 0 TO nTempIolByteLength - 1 DO
		IF nComplex > cBASIC_TYPE THEN
			aTempValues[nTempIndex] := aTempItems[nTempIolByteLength - 1 - nTempIndex];
		ELSE
			aTempValues[nTempIndex] := aIolRecords[nTempIolByteLength - 1 - nTempIndex];
		END_IF;
	END_FOR;	  	 
	  	
// Copy result into a DWORD variable
	F_Leuze_IOL_GetInteger := PDWORD_TO_DWORD(ADR(aTempValues));
	  
// Received value can be a negative value
	IF bIsSigned THEN
	// Create a signed value
		IF DWORD_TO_BOOL(SHR(F_Leuze_IOL_GetInteger, INT_TO_UINT(nBitLength) - 1)) THEN
			nTemp := 2;
			FOR nTempIndex := 1 TO nBitLength - 1 DO
				nTemp := nTemp * 2;
			END_FOR;
			F_Leuze_IOL_GetInteger := F_Leuze_IOL_GetInteger OR (16#FFFF_FFFF XOR (nTemp - 1));
			END_IF;
		END_IF;
	END_IF;

END_FUNCTION

// Leuze/Internal/F_Leuze_IOL_GetString
FUNCTION F_Leuze_IOL_GetString : STRING
VAR_INPUT 
      nComplex : INT;	// Data type: cBASIC_TYPE, cCOMPLEX_RECORD_TYPE, cCOMPLEX_ARRAY_TYPE
      nComplexDataTypeSize : INT;	// Record or Array type size
      nOffset : INT;	// Bit Offset
      nFixedLength : INT; // In bits
   END_VAR
   VAR_IN_OUT 
      aIolRecords : ARRAY[0..cNUMBER_IOLINK_DATA] OF BYTE;
      aTempItems : ARRAY[0..cNUMBER_IOLINK_DATA] OF BYTE;
   END_VAR
   VAR 
      nTempIndex : INT;
	  nTempStringLength : UINT;
	  nTempByteLength : INT;
   END_VAR
   VAR CONSTANT 
	cNUMBER_IOLINK_DATA : INT := 255;   //   Number of IO Link record data
	cBITS_IN_BYTE : INT := 8;   //   Number of bits in byte
	cBASIC_TYPE : INT := 0;
	cCOMPLEX_RECORD_TYPE : INT := 1;
	cCOMPLEX_ARRAY_TYPE : INT := 2;
END_VAR

// =============================================================================
	// Name:    IO-Link internal function 
	//          Get string
	// Date:    01.07.2020
	// ==============================================================================	
	//Data type is part of a Record data type
	IF nComplex = cCOMPLEX_RECORD_TYPE THEN
	  F_Leuze_IOL_GetRecordT( nComplexDataTypeSize, nOffset, nFixedLength, aIolRecords, aTempItems);
	//Data type is part of a Array data type
	ELSIF nComplex = cCOMPLEX_ARRAY_TYPE THEN
	  F_Leuze_IOL_GetArrayT(INT_TO_UINT(nComplexDataTypeSize), INT_TO_UINT(nOffset), INT_TO_UINT(nFixedLength), aIolRecords, aTempItems);
	END_IF;
	
	//Initialization
	nTempStringLength := 0;
	nTempByteLength := nFixedLength / cBITS_IN_BYTE;

	//Calculate the actual string length
	IF nTempByteLength <= 232 THEN
	  FOR nTempIndex := 0 TO nTempByteLength - 1 DO
	    IF nComplex > 0 THEN
	      IF aTempItems[nTempIndex] = 16#00 THEN
	        EXIT;
	      ELSE
	        nTempStringLength := nTempStringLength + 1;
	      END_IF;
	    ELSE
	      IF aIolRecords[nTempIndex] = 16#00 THEN
	        EXIT;
	      ELSE
	        nTempStringLength := nTempStringLength + 1;
	      END_IF;
	    END_IF;
	  END_FOR;
	  
	  //Copy to the RETURN value
	  IF nComplex > cBASIC_TYPE THEN		  		   
		  F_Leuze_IOL_GetString := BYTEARR_TO_MAXSTRING(aTempItems);		  
	  ELSE
	    IF nTempStringLength = 0 THEN
	      F_Leuze_IOL_GetString := '';
	    ELSE
			F_Leuze_IOL_GetString := BYTEARR_TO_MAXSTRING(aIolRecords);
	    END_IF;
	  END_IF;
	ELSE
	  F_Leuze_IOL_GetString := '';
	END_IF;

END_FUNCTION

// Leuze/Internal/F_Leuze_IOL_SetArrayT
FUNCTION F_Leuze_IOL_SetArrayT : BOOL
VAR_INPUT 
      nArraySize : UINT;
      nItemPosition : UINT;
      nBitLength : UINT;
   END_VAR
   VAR_IN_OUT 
      aIolRecords : ARRAY[0..cNUMBER_IOLINK_DATA] OF BYTE;
      aTempItems : ARRAY[0..cNUMBER_IOLINK_DATA] OF BYTE;
   END_VAR
   VAR
      nTempArrayByteLength : UINT;
      nTempStartByte : UINT;
      nTempStartBit : UINT;
      nTempIolBitLength : UINT;
      nTempIndex : UINT;
      nTempShiftByte : BYTE;
      bTempByteFill : BOOL;
   END_VAR
   VAR CONSTANT 
	  cNUMBER_IOLINK_DATA : UINT := 255;   //   Number of IO Link record data
	  cBITS_IN_BYTE : UINT := 8;   //   Number of bits in byte
   END_VAR

// =============================================================================
// Name:    IO-Link internal function 
//	 	    Set ArrayT
// Date:    01.01.2021
// ==============================================================================
	
// Initialize variables
	bTempByteFill := FALSE;
	nTempIndex := 0;

// Bit length of the current item
	nTempIolBitLength := nBitLength;

// Get byte length of the whole array
	nTempArrayByteLength := F_Leuze_IOL_GetByteLength(nArraySize);
	
// Calculate the start byte of the current array item
	nTempStartByte := nTempArrayByteLength - 1 - ((nArraySize - (nItemPosition * nTempIolBitLength)) / cBITS_IN_BYTE);
	
// Calculate the start bit of the current array item
	nTempStartBit := (nArraySize - (nItemPosition * nTempIolBitLength)) MOD cBITS_IN_BYTE;
	
// Set array item
	WHILE nTempIolBitLength > 0 DO
	  IF NOT bTempByteFill THEN
	    IF (nTempIolBitLength + nTempStartBit) < cBITS_IN_BYTE THEN
	      nTempShiftByte := SHL(aTempItems[nTempIndex], cBITS_IN_BYTE - nTempIolBitLength);
	      nTempShiftByte := SHR(nTempShiftByte, (cBITS_IN_BYTE - nTempIolBitLength) - nTempStartBit);
	    ELSE
	      nTempShiftByte := SHL(aTempItems[nTempIndex], nTempStartBit);
	    END_IF;
	    
	    aIolRecords[nTempStartByte] := aIolRecords[nTempStartByte] + nTempShiftByte;
	    
	    IF (nTempStartBit + nTempIolBitLength) = cBITS_IN_BYTE THEN
	      nTempStartByte := nTempStartByte - 1;
	    END_IF;
	    
	    IF (nTempStartBit + nTempIolBitLength) > cBITS_IN_BYTE THEN
	      nTempStartByte := nTempStartByte - 1;
	      bTempByteFill := TRUE;
	    ELSE
	      nTempIndex := nTempIndex + 1;
	    END_IF;
	    
	    nTempIolBitLength := nTempIolBitLength - (cBITS_IN_BYTE - nTempStartBit);
	  ELSE
	    IF nTempStartBit > nTempIolBitLength THEN
	      nTempShiftByte := SHL(aTempItems[nTempIndex], nTempStartBit - nTempIolBitLength);
	      nTempShiftByte := SHR(nTempShiftByte, cBITS_IN_BYTE - nTempIolBitLength);
	    ELSE
	      nTempShiftByte := SHR(aTempItems[nTempIndex], cBITS_IN_BYTE - nTempStartBit);
	    END_IF;
	    
	    aIolRecords[nTempStartByte] := aIolRecords[nTempStartByte] + nTempShiftByte;
	    nTempIolBitLength := nTempIolBitLength - nTempStartBit;
	    nTempIndex := nTempIndex + 1;
	    bTempByteFill := FALSE;
	  END_IF;
	END_WHILE;

END_FUNCTION

// Leuze/Internal/F_Leuze_IOL_SetBoolean
FUNCTION F_Leuze_IOL_SetBoolean : BOOL
VAR_INPUT 
      nComplex : INT;	// Data type: cBASIC_TYPE, cCOMPLEX_RECORD_TYPE, cCOMPLEX_ARRAY_TYPE
      nComplexDataTypeSize : INT;	// Record or Array type size
      nOffset : INT;	// Bit Offset
      bSource : BOOL;
   END_VAR
   VAR_IN_OUT 
      aIolRecords : ARRAY[0..cNUMBER_IOLINK_DATA] OF BYTE;
      aTempItems : ARRAY[0..cNUMBER_IOLINK_DATA] OF BYTE;
   END_VAR
   VAR CONSTANT 
      cNUMBER_IOLINK_DATA : INT := 255;   //   Number of IO Link record data
      cBASIC_TYPE : INT := 0;
      cCOMPLEX_RECORD_TYPE : INT := 1;
      cCOMPLEX_ARRAY_TYPE : INT := 2;
   END_VAR

// =============================================================================
// Name:    IO-Link internal function 
//          Set Boolean
// Date:    01.07.2020
// ==============================================================================
// In a nComplex data type the coding of booleans are only 1 bit wide. There is no padding to byte
IF nComplex > cBASIC_TYPE THEN
  IF bSource THEN
    aTempItems[0] := (aTempItems[0] AND 2#1111_1110) + 1;
  ELSE
    aTempItems[0] := aTempItems[0] AND 2#1111_1110;
  END_IF;
ELSE
  IF bSource THEN
    aIolRecords[0] := 16#FF;
  ELSE
    aIolRecords[0] := 16#00;
  END_IF;
END_IF;

// Data type is part of a Record data type
IF nComplex = cCOMPLEX_RECORD_TYPE THEN
  F_Leuze_IOL_SetRecordT(nComplexDataTypeSize, nOffset, 1, aIolRecords, aTempItems);
// Data type is part of a Array data type
ELSIF nComplex = cCOMPLEX_ARRAY_TYPE THEN
  F_Leuze_IOL_SetArrayT(INT_TO_UINT(nComplexDataTypeSize), INT_TO_UINT(nOffset), 1, aIolRecords, aTempItems);
END_IF;

END_FUNCTION

// Leuze/Internal/F_Leuze_IOL_SetRecordT
FUNCTION F_Leuze_IOL_SetRecordT : BOOL
VAR_INPUT 
      nRecordSize : INT;
      nBitOffset : INT;
      nBitLength : INT;
   END_VAR
   VAR_IN_OUT 
      aIolRecords : ARRAY[0..cNUMBER_IOLINK_DATA] OF BYTE;
      aTempItems : ARRAY[0..cNUMBER_IOLINK_DATA] OF BYTE;
   END_VAR
   VAR 
      nTempStartByte : INT;
      nTempStartBit : INT;
      nTempIolBitLength : INT;
      nTempIndex : INT;
      nTempShiftByte : BYTE;
      bTempByteFill : BOOL;
   END_VAR
   VAR CONSTANT 
	  cNUMBER_IOLINK_DATA : INT := 255;   //   Number of IO Link record data
	  cBITS_IN_BYTE : INT := 8;   //   Number of bits in byte
   END_VAR

//=============================================================================
	//Name:    IO-Link internal function 
	//		   Set RecordT
	//Date:    01.07.2020
	//==============================================================================
	
	//Initialize variables
	bTempByteFill := FALSE;
	nTempIndex := 0;
	
	//Bit length of the current item
	nTempIolBitLength := nBitLength;
	
	// Calculate the start byte of the current item
	nTempStartByte := (nRecordSize / cBITS_IN_BYTE) - 1 - (nBitOffset / cBITS_IN_BYTE);
	IF NOT(nRecordSize MOD cBITS_IN_BYTE = 0) THEN
		nTempStartByte := nTempStartByte + 1;
	END_IF;
	
	//Calculate the start bit of the current item
	nTempStartBit := nBitOffset MOD cBITS_IN_BYTE;
	
	//Set record item
	WHILE nTempIolBitLength > 0 DO
	  IF NOT bTempByteFill THEN
	    IF (nTempIolBitLength + nTempStartBit) < cBITS_IN_BYTE THEN
	      nTempShiftByte := SHL(aTempItems[nTempIndex], INT_TO_UINT(cBITS_IN_BYTE - nTempIolBitLength));
	      nTempShiftByte := SHR(nTempShiftByte, INT_TO_UINT((cBITS_IN_BYTE - nTempIolBitLength) - nTempStartBit));
	    ELSE
	      nTempShiftByte := SHL(aTempItems[nTempIndex], INT_TO_UINT(nTempStartBit));
	    END_IF;
	    
	    aIolRecords[nTempStartByte] := aIolRecords[nTempStartByte] + nTempShiftByte;
	    
	    IF (nTempStartBit + nTempIolBitLength) = cBITS_IN_BYTE THEN
	      nTempStartByte := nTempStartByte - 1;
	    END_IF;
	    
	    IF (nTempStartBit + nTempIolBitLength) > cBITS_IN_BYTE THEN
	      nTempStartByte := nTempStartByte - 1;
	      bTempByteFill := TRUE;
	    ELSE
	      nTempIndex := nTempIndex + 1;
	    END_IF;
	    
	    nTempIolBitLength := nTempIolBitLength - (cBITS_IN_BYTE - nTempStartBit);
	  ELSE
	    IF nTempStartBit > nTempIolBitLength THEN
	      nTempShiftByte := SHL(aTempItems[nTempIndex], INT_TO_UINT(nTempStartBit - nTempIolBitLength));
	      nTempShiftByte := SHR(nTempShiftByte, INT_TO_UINT(cBITS_IN_BYTE - nTempIolBitLength));
	    ELSE
	      nTempShiftByte := SHR(aTempItems[nTempIndex], INT_TO_UINT(cBITS_IN_BYTE - nTempStartBit));
	    END_IF;
	    
	    aIolRecords[nTempStartByte] := aIolRecords[nTempStartByte] + nTempShiftByte;
	    nTempIolBitLength := nTempIolBitLength - nTempStartBit;
	    nTempIndex := nTempIndex + 1;
	    bTempByteFill := FALSE;
	  END_IF;
	END_WHILE;

END_FUNCTION

// Leuze/Internal/F_Leuze_IOL_SetInteger
FUNCTION F_Leuze_IOL_SetInteger : BOOL
VAR_INPUT 
      nComplex : INT;	// Data type: cBASIC_TYPE, cCOMPLEX_RECORD_TYPE, cCOMPLEX_ARRAY_TYPE
      nComplexDataTypeSize : INT;	// Record or Array type size
      nOffset : INT;	// Bit Offset
      nSource : DWORD;
      nBitLength : INT;
   END_VAR
   VAR_IN_OUT 
      aIolRecords : ARRAY[0..cNUMBER_IOLINK_DATA] OF BYTE;
      aTempItems : ARRAY[0..cNUMBER_IOLINK_DATA] OF BYTE;
   END_VAR
   VAR
      nTempIndex : INT;
      nTempIolByteLength : INT;
	  pByte: POINTER TO BYTE;
      aTempValues : ARRAY[0..3] OF BYTE;
   END_VAR
   VAR CONSTANT 
	  cNUMBER_IOLINK_DATA : INT := 255;   //   Number of IO Link record data
	  cBITS_IN_BYTE : INT := 8;   //   Number of bits in byte
      cBASIC_TYPE : INT := 0;
      cCOMPLEX_RECORD_TYPE : INT := 1;
      cCOMPLEX_ARRAY_TYPE : INT := 2;
   END_VAR

// =============================================================================
// Name:    IO-Link internal function 
//    		Set Integer
// Date:    01.07.2020
// ==============================================================================

// Get byte length
	nTempIolByteLength := nBitLength / cBITS_IN_BYTE;
	IF NOT (nBitLength MOD cBITS_IN_BYTE = 0) THEN
		nTempIolByteLength := nTempIolByteLength + 1;
	END_IF;

// There is no padding to 1,2,4 byte if a nComplex data type is used
	IF (nComplex = cBASIC_TYPE) AND (nTempIolByteLength = 3) THEN
		nTempIolByteLength := 4;
	END_IF;

	IF nTempIolByteLength > 0 AND nTempIolByteLength <= 4 THEN
		pByte := ADR(nSource);
		// Copy value
		IF nTempIolByteLength = 1 THEN
			aTempValues[0] := pByte[0];
			aTempValues[1] := 0;
			aTempValues[2] := 0;
			aTempValues[3] := 0;
		ELSIF nTempIolByteLength = 2 THEN
			aTempValues[0] := pByte[1];
			aTempValues[1] := pByte[0];
			aTempValues[2] := 0;
			aTempValues[3] := 0;		
		ELSIF nTempIolByteLength = 4 THEN
			aTempValues[3] := pByte[0];
			aTempValues[2] := pByte[1];
			aTempValues[1] := pByte[2];			
			aTempValues[0] := pByte[3];					
		END_IF;
		
		// Is part of an record or an array data type
		IF nComplex > cBASIC_TYPE THEN
		FOR nTempIndex := 0 TO nTempIolByteLength - 1 DO
			aTempItems[nTempIndex] := aTempValues[nTempIolByteLength - 1 - nTempIndex];
		END_FOR;
		
		// Is a simple data type
		ELSE
		FOR nTempIndex := nTempIolByteLength - 1 TO 0 BY -1 DO
			aIolRecords[nTempIndex] := aTempValues[nTempIndex];
		END_FOR;
		END_IF;
		
		// Data type is part of a Record data type
		IF nComplex = cCOMPLEX_RECORD_TYPE THEN
			F_Leuze_IOL_SetRecordT(nComplexDataTypeSize, nOffset, nBitLength, aIolRecords, aTempItems);
		// Data type is part of a Array data type
		ELSIF nComplex = cCOMPLEX_ARRAY_TYPE THEN
			F_Leuze_IOL_SetArrayT(INT_TO_UINT(nComplexDataTypeSize), INT_TO_UINT(nOffset), INT_TO_UINT(nBitLength), aIolRecords, aTempItems);
		END_IF;
	END_IF;

END_FUNCTION

// Leuze/Internal/F_Leuze_IOL_SetString
FUNCTION F_Leuze_IOL_SetString : BOOL
VAR_INPUT 
      nComplex : INT;	// Data type: cBASIC_TYPE, cCOMPLEX_RECORD_TYPE, cCOMPLEX_ARRAY_TYPE
      nComplexDataTypeSize : INT;	// Record or Array type size
      nOffset : INT;	// Bit Offset
      nFixedLength : INT; // In bites
      sSource : String;
   END_VAR
   VAR_IN_OUT 
      aIolRecords : ARRAY[0..cNUMBER_IOLINK_DATA] OF BYTE;
      aTempItems : ARRAY[0..cNUMBER_IOLINK_DATA] OF BYTE;
   END_VAR
   VAR 
	  nTempIndex : INT;
	  nTempByteLength : INT;
      nTempStringLength : INT;
      aTempValues : ARRAY[0..255] OF BYTE;
   END_VAR
   VAR CONSTANT 
	cNUMBER_IOLINK_DATA : INT := 255;   //   Number of IO Link record data
	cBITS_IN_BYTE : INT := 8;   //   Number of bits in byte
	cBASIC_TYPE : INT := 0;
	cCOMPLEX_RECORD_TYPE : INT := 1;
	cCOMPLEX_ARRAY_TYPE : INT := 2;
 END_VAR

// =============================================================================
// Name:    IO-Link internal function 
//          Set string
// Date:    01.07.2020
// ==============================================================================

//Initialization
nTempByteLength := nFixedLength / cBITS_IN_BYTE;

//Copy input data
aTempValues := MAXSTRING_TO_BYTEARR(sSource);

//Get string length
nTempStringLength := LEN(sSource);

IF nTempByteLength > 0 AND nTempByteLength <= UDINT_TO_INT(MAX_STRING_LENGTH) THEN
    //Is part of an record or an array data type
    IF nComplex > cBASIC_TYPE THEN
    FOR nTempIndex := 0 TO nTempByteLength - 1 DO
        IF nTempStringLength < nTempByteLength - nTempIndex THEN
        aTempItems[nTempIndex] := 16#00;
        ELSE
        aTempItems[nTempIndex] := aTempValues[nTempByteLength - 1 - nTempIndex];
        END_IF;
    END_FOR;
    
    //Is a simple data type
    ELSE
    FOR nTempIndex := 0 TO nTempByteLength - 1 DO
        IF nTempIndex <= nTempStringLength - 1 THEN
        aIolRecords[nTempIndex] := aTempValues[nTempIndex];
        ELSE
        aIolRecords[nTempIndex] := 16#00;
        END_IF;
    END_FOR;
    END_IF;
    
    //Data type is part of a Record data type
    IF nComplex = cCOMPLEX_RECORD_TYPE THEN
    	F_Leuze_IOL_SetRecordT(nComplexDataTypeSize, nOffset, nFixedLength, aIolRecords, aTempItems);
    //Data type is part of a Array data type
    ELSIF nComplex = cCOMPLEX_ARRAY_TYPE THEN
    	F_Leuze_IOL_SetArrayT(INT_TO_UINT(nComplexDataTypeSize), INT_TO_UINT(nOffset), INT_TO_UINT(nFixedLength), aIolRecords, aTempItems);
    END_IF;
END_IF;

END_FUNCTION

// Leuze/Internal/F_Leuze_IOL_SortComplex
FUNCTION F_Leuze_IOL_SortComplex : BOOL
VAR_INPUT 
      nComplex : INT;	// Data type: cBASIC_TYPE, cCOMPLEX_RECORD_TYPE, cCOMPLEX_ARRAY_TYPE
      nComplexDataTypeSize : INT;	// Record or Array type size
      nOffset : INT;	// Bit Offset
      nBitLength : INT;	
   END_VAR
   VAR_IN_OUT 
      aIolRecords : ARRAY[0..cNUMBER_IOLINK_DATA] OF BYTE;
      aTempItems : ARRAY[0..cNUMBER_IOLINK_DATA] OF BYTE;
   END_VAR
   VAR CONSTANT 
      cNUMBER_IOLINK_DATA : INT := 255;   //   Number of IO Link record data
      cBASIC_TYPE : INT := 0;
      cCOMPLEX_RECORD_TYPE : INT := 1;
      cCOMPLEX_ARRAY_TYPE : INT := 2;
   END_VAR

//=============================================================================
//Name:    IO-Link internal function 
//Date:    01.07.2020
//==============================================================================
	
//Data type is part of a Record data type
IF nComplex = cCOMPLEX_RECORD_TYPE THEN
  F_Leuze_IOL_GetRecordT(nComplexDataTypeSize, nOffset, nBitLength, aIolRecords, aTempItems);
//Data type is part of a Array data type
ELSIF nComplex = cCOMPLEX_ARRAY_TYPE THEN
  F_Leuze_IOL_GetArrayT(nComplexDataTypeSize, nOffset, nBitLength, aIolRecords, aTempItems);
END_IF;

//Set IO-Link record data
IF nComplex = cBASIC_TYPE THEN
  aTempItems := aIolRecords;
END_IF;

END_FUNCTION

// Leuze/Internal/FB_Leuze_IOL_AdsReadWrite
FUNCTION_BLOCK FB_Leuze_IOL_AdsReadWrite
VAR_INPUT
	bExecute : BOOL;   // Positive trigger: Start data transfer
	// String containing the AMS network identifier of the target device to which the ADS command is directed
	sNetID: T_AmsNetID;
	//  Port number of the ADS device
	nPort: T_AmsPort;
	//  Index group number
	nIdxGroup: UDINT;
	// Index of the IODD parameter
	nIndex: INT;
	// Subindex of the IODD parameter
	nSubIndex: INT;
	// Number, in bites, of the data to be read.
	nLen: UINT;
END_VAR
VAR_STAT
      // Read or write the selected IO-Link parameter. The ADS command is triggered by a rising edge at this input. 
	// FALSE: Read parameter
	// TRUE: Write Parameter
	bStatRW : BOOL;
END_VAR
VAR_INPUT
      // Read or write the selected IO-Link parameter. The ADS command is triggered by a rising edge at this input. 
	// FALSE: Read parameter
	// TRUE: Write Parameter
	bRW : BOOL;
    tTimeOut : TIME := DEFAULT_ADS_TIMEOUT;   // Time, after a Timeout-Error is triggered.
END_VAR
VAR_IN_OUT
	// Data to be written or read.
	aData: ARRAY[0..cNUMBER_IOLINK_DATA] OF BYTE;
END_VAR
VAR_OUTPUT
	bValid : BOOL;   // Indicates whether data is valid.
    bBusy  : BOOL;   // Request in process. FALSE: Request is terminated TRUE: Request is being processed
    bError  : BOOL;   // Error flag FALSE: No error TRUE: Error detected
    stErrorCode : ST_Leuze_IOL_Error;   // Status of the function block
	// Number of successfully read data bytes.
	nCount: UINT;
END_VAR
VAR
	// Block for executing an ADS write command for transferring data to an ADS device.
	fbWriteReq: ADSWRITE;
	// The function block executes an ADS read command to request data from an ADS device.
	fbReadReq  : ADSREADEX;
END_VAR
VAR_STAT
	nStatLen: UDINT;
    bStatBusyMem : BOOL;
    bStatTriggerExecute : BOOL;
    bStatTriggerExecuteMem : BOOL;
	bStatError: BOOL;
	bStatBusy: BOOL;
	stStatErrorCode: ST_Leuze_IOL_Error;
    aStatIOLRecords : ARRAY[0..cNUMBER_IOLINK_DATA] OF BYTE;
	nStatCount: UDINT;
	nStatState: INT;
	nStatIndexOffset: UDINT;
END_VAR
VAR CONSTANT
    cDEFAULT : WORD := 16#0000;   // Order completed, no warning or further detailing
	// bError: ADS read/write
	cERR_ADS_READ_WRITE: WORD := 16#8003;
    cERR_TIME_OUT : WORD := 16#8001;   // Error: Time out detected
	// Init
	cSTATE_INIT: INT := 1;
	// Send request
	cSTATE_RW: INT := 2;
	// Wait for response
	cSTATE_RESPONSE: INT := 3;
	// Job done
	cSTATE_JOB_DONE: INT := 4;
    cBITS_IN_BYTE : UINT := 8;   // Number of bits in byte
	cINDEX_BIT_SHIFT: INT := 16;
    cNUMBER_IOLINK_DATA : INT := 255;   // Number of IO Link record data
END_VAR
VAR_TEMP
	// temp loop indexer
	nTempLoopIndex: INT;
END_VAR

//=============================================================================
//Name:                 FB_Leuze_AdsReadWrite
//Company:              Leuze electronic GmbH + Co.KG
//Date:                 01.01.2021
//Version:    			V1.0.0
//-----------------------------------------------------------------------------

//Init
	bStatTriggerExecute := bExecute AND NOT bStatTriggerExecuteMem;
	bStatTriggerExecuteMem := bExecute;
	IF bStatTriggerExecute AND NOT bStatBusyMem THEN
		nStatState := cSTATE_INIT;
	END_IF
CASE nStatState  OF
	cSTATE_INIT:		
		bStatBusyMem := TRUE;
		bValid := FALSE;
		bBusy := TRUE;
		// IndexOffset = index 16bits subindex 16bits
		nStatIndexOffset := INT_TO_UDINT(nIndex);
		nStatIndexOffset := SHL(nStatIndexOffset, cINDEX_BIT_SHIFT);
		nStatIndexOffset := nStatIndexOffset OR INT_TO_UDINT(nSubIndex);
		nStatLen := F_Leuze_IOL_GetByteLength(nLen);
		bError := FALSE;	        
		stErrorCode.nBlockError := cDEFAULT;
		stErrorCode.nAdsReadError := cDEFAULT;
		stErrorCode.nAdsWriteError := cDEFAULT;
		stErrorCode.nIndex := 0;
		stErrorCode.nSubIndex := 0;
		aStatIOLRecords := aData;
		bStatRW := bRW;		
		IF bStatRW THEN
			fbWriteReq( WRITE := TRUE, NETID := sNetID, PORT := nPort, IDXGRP := nIdxGroup,  IDXOFFS := nStatIndexOffset, LEN := nStatLen, TMOUT := tTimeOut, SRCADDR := ADR(aStatIOLRecords));
		ELSE
			FOR nTempLoopIndex := 0 TO cNUMBER_IOLINK_DATA DO
	        	aStatIOLRecords[nTempLoopIndex] := 16#00;
	        END_FOR;
			fbReadReq( READ := TRUE, NETID := sNetID, PORT := nPort, IDXGRP := nIdxGroup, IDXOFFS := nStatIndexOffset, LEN := nStatLen , TMOUT := tTimeOut, DESTADDR := ADR(aStatIOLRecords));
		END_IF				
		nStatState := cSTATE_RW;		

	cSTATE_RW:
		IF bStatRW THEN
			fbWriteReq(BUSY => bStatBusy, ERR => bStatError, ERRID => stStatErrorCode.nAdsWriteError);
		ELSE
			fbReadReq(BUSY => bStatBusy, ERR => bStatError, ERRID => stStatErrorCode.nAdsReadError, COUNT_R => nStatCount);
		END_IF
		IF bStatBusyMem AND NOT bStatBusy THEN	
			fbWriteReq(WRITE := FALSE);
			fbReadReq(READ := FALSE);
			nStatState := cSTATE_RESPONSE;
		END_IF
		
	cSTATE_RESPONSE:				
		bBusy := FALSE;
		bStatBusyMem := FALSE;		
		IF bStatError THEN
			bError := TRUE;
			stErrorCode.nBlockError := cERR_ADS_READ_WRITE;
			stErrorCode.nAdsReadError := stStatErrorCode.nAdsReadError;
			stErrorCode.nAdsWriteError := stStatErrorCode.nAdsWriteError;	            
			stErrorCode.nIndex := nIndex;
			stErrorCode.nSubIndex := nSubIndex;
		ELSE
			bValid := TRUE;
			nCount := UDINT_TO_UINT(nStatCount) * cBITS_IN_BYTE;
			aData := aStatIOLRecords;				
		END_IF	
		nStatState := cSTATE_JOB_DONE;					
END_CASE

END_FUNCTION_BLOCK

// Leuze/F_Leuze_PD_DMU218_3091
FUNCTION F_Leuze_PD_DMU218_3091 : ST_Leuze_PD_DMU218_3091	// Reference to the instance of the data structure ST_Leuze_PD_DMU218_3091. The structure includes the disaggregated values of the process data.
VAR_INPUT
	aProcessData : ARRAY[0..1] OF BYTE;    // Raw process data of the IO-Link device.
END_VAR
VAR_OUTPUT
	bError : BOOL;    // Error flag FALSE: No error TRUE: Error detected
END_VAR
VAR
	aTempIOLRecords : ARRAY[0..cNUMBER_IOLINK_DATA] OF BYTE;
	aTempTempItems : ARRAY[0..cNUMBER_IOLINK_DATA] OF BYTE;
	nTempCopyResult : UDINT;
	stTempSensorData : ST_Leuze_PD_DMU218_3091;
	stTempOutputSensorData : ST_Leuze_PD_DMU218_3091;
END_VAR
VAR CONSTANT
	cCOMPLEX_RECORD_TYPE : INT := 1;    // IODD data type - RecordT
	cCOMPLEX_ARRAY_TYPE : INT := 2;    // IODD data type - ArrayT
	cBASIC_TYPE : INT := 0;    // IODD data type - BasicT - BoolT, UIntegerT, ...
	cBITS_IN_BYTE : INT := 8;    // Number of bits in byte
	cNUMBER_PD_DATA : UDINT := 2;    // Length of PD data in bytes
	cNUMBER_IOLINK_DATA : INT := 255;    // Number of IO Link record data
END_VAR

//=============================================================================
//Name:                 F_Leuze_PD_DMU218_3091
//Company:              Leuze electronic GmbH + Co.KG
//Date:                 04/09/2023
//Generator Version:    V3.3.0.0
//IODD Version:         V1.2
//IODD Release date:    20230801
//-----------------------------------------------------------------------------

//Copy process data
	nTempCopyResult:= MEMMOVE(ADR(aTempIOLRecords), ADR(aProcessData), cNUMBER_PD_DATA);
	IF nTempCopyResult = 0 THEN
		bError := TRUE;
		RETURN;
	ELSE
		bError := FALSE;
	END_IF;

//Assign new values to output
	stTempOutputSensorData.nMeasuredValue := DWORD_TO_UINT(F_Leuze_IOL_GetInteger(nComplex := cCOMPLEX_RECORD_TYPE, nComplexDataTypeSize := 16, nOffset := 4, nBitLength := 12, bIsSigned := False, aIolRecords := aTempIolRecords, aTempItems := aTempTempItems));
	stTempOutputSensorData.bSwitchStateBdc1Q1 := F_Leuze_IOL_GetBoolean(nComplex := cCOMPLEX_RECORD_TYPE, nComplexDataTypeSize := 16, nOffset := 0, aIolRecords := aTempIolRecords, aTempItems := aTempTempItems);

// Return
	F_Leuze_PD_DMU218_3091 := stTempOutputSensorData;

END_FUNCTION

// Leuze/FB_Leuze_IOL_DMU218_3091
FUNCTION_BLOCK FB_Leuze_IOL_DMU218_3091
VAR_INPUT
	bExecute : BOOL;    // Positive trigger: Start data transfer
	sNetID : T_AmsNetID;	// String containing the AMS network identifier of the target device to which the ADS command is directed.
	nPort : T_AmsPort;	// Port number of the ADS device.
	nIdxGroup : UDINT;    // Index group number
	bRW : BOOL;    // Read or write the selected IO-Link parameter. FALSE: Read parameter TRUE: Write Parameter.
	tTimeOut : TIME;    // Time, after a Timeout-Error is triggered.
END_VAR
VAR_IN_OUT
	stDeviceData : ST_Leuze_IOL_DMU218_3091;	// SensorData
END_VAR
VAR_OUTPUT
	bDone : BOOL;    // Indicates whether data is valid.
	bBusy : BOOL;    // Request in process. FALSE: Request is terminated TRUE: Request is being processed
	bError : BOOL;    // Error flag FALSE: No error TRUE: Error detected
	stErrorCode : ST_Leuze_IOL_Error;	// Status of the function block
END_VAR
VAR
	fbReadWriteReq : FB_Leuze_IOL_AdsReadWrite;
END_VAR
VAR_TEMP
	nTempLoopIndex : INT;    // Loop indexer
	bTempDeviceDataBOOL : BOOL;    // Temporary memory for data conversion
	nTempDeviceDataInteger : DWORD;    // Temporary memory for data conversion
	sTempDeviceDataString : STRING;    // Temporary memory for data conversion
END_VAR
VAR_STAT
	bStatTriggerDone : BOOL;
	bStatTriggerError : BOOL;
	bStatTriggerExecute : BOOL;
	bStatTriggerDoneMem : BOOL;
	bStatTriggerErrorMem : BOOL;
	bStatTriggerExecuteMem : BOOL;
	bStatBusyMem : BOOL;
	bStatRWSave : BOOL;
	nStatIndex : USINT;
	nStatElement : INT;    // Element of complex data type
	nStatState : INT;    // State of the job
	nStatNumSelection : INT;
	nStatCommandIndex : INT;
	bStatSource : BOOL;
	nStatComplex : INT;    // IODD data type: basic, record, array
	nStatComplexDataTypeSize : INT;
	nStatOffset : INT;
	nStatBitLength : UINT;    // Length of the data type in bits
	stStatLastErrorCode : ST_Leuze_IOL_Error;	// ST_Leuze_IOL_Error
	fbInstTimeOut : TON;
	aStatInputSelections : ARRAY[0..cNUMBER_INPUTS] OF BOOL;
	aStatIOLRecords : ARRAY[0..cNUMBER_IOLINK_DATA] OF BYTE;
	aStatCommandQueue : ARRAY[0..cNUMBER_IOLINK_DATA] OF ST_Leuze_IOL_CommandQueue;
	aStatTempItems : ARRAY[0..cNUMBER_IOLINK_DATA] OF BYTE;
END_VAR
VAR CONSTANT
	cSTATE_READY : INT := 0;
	cSTATE_INIT : INT := 1;    // State parsing input selection
	cSTATE_CLEAR_RECORD : INT := 2;    // State clearing data record
	cSTATE_SEND_REQUEST : INT := 3;    // State sending request
	cSTATE_AWAIT_RESPONSE : INT := 4;    // State waiting for response
	cSTATE_PARSE_RESPONSE : INT := 5;    // State parsing response
	cSTATE_JOB_FINISHED : INT := 6;    // State job finished
	cCOMPLEX_RECORD_TYPE : INT := 1;    // IODD data type - RecordT
	cCOMPLEX_ARRAY_TYPE : INT := 2;    // IODD data type - ArrayT
	cBASIC_TYPE : INT := 0;    // IODD data type - BasicT - BoolT, UINTegerT, ...
	cBITS_IN_BYTE : INT := 8;    // Number of bits in byte
	cDEFAULT : WORD := 16#0000;    // Order completed, no warning or further detailing
	cERR_TIME_OUT : WORD := 16#8001;    // Error: Time out detected
	cERR_EMPTY_SELECTION : WORD := 16#8200;    // Error: No parameter selected
	cNUMBER_IOLINK_DATA : INT := 255;    // Number of IO Link record data
	cEMPTY_COMMAND_QUEUE : INT := -1;    // Empty command queue
	cNUMBER_INPUTS : INT := 100;    // Index of last input parameter
END_VAR

//=============================================================================
//Name:                 FB_Leuze_IOL_DMU218_3091
//Company:              Leuze electronic GmbH + Co.KG
//Date:                 04/09/2023
//Generator Version:    V3.3.0.0
//IODD Version:         V1.1
//IODD Release date:    20230801
//-----------------------------------------------------------------------------

